FUNCTION_BLOCK IL (* Input service interface function block for long word input data *)
  (* Description: Copyright (c) 2018 TU Wien/ACIN This program and the accompanying materials are made available under the terms of the Eclipse Public License 2.0 which is available at https://www.eclipse.org/legal/epl-2.0/ SPDX-License-Identifier: EPL-2.0 *)
  (* Version 3.0, 2025-04-14, Patrick Aigner, changed package *)
  (* Version 1.0, 2018-10-05, Martin Melik-Merkumians, TU Wien/ACIN *)
  PACKAGE eclipse4diac::io;
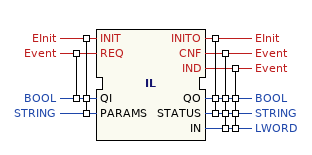
  EVENT_INPUT
    INIT : EInit WITH QI, PARAMS; (* Service Initialization *)
    REQ WITH QI; (* Service Request *)
  END_EVENT
  EVENT_OUTPUT
    INITO : EInit WITH QO, STATUS; (* Initialization Confirm *)
    CNF WITH QO, STATUS, IN; (* Confirmation of Requested Service *)
    IND WITH QO, STATUS, IN; (* Indication from Resource *)
  END_EVENT
  VAR_INPUT
    QI : BOOL; (* Event Input Qualifier *)
    PARAMS : STRING; (* Service Parameters *)
  END_VAR
  VAR_OUTPUT
    QO : BOOL; (* Event Output Qualifier *)
    STATUS : STRING; (* Service Status *)
    IN : LWORD; (* Input data from resource *)
  END_VAR
END_FUNCTION_BLOCK
